// TIA Portal V18 export
// export: Created 2023-08-22T11:16:04.1404114Z, ExportSetting WithDefaults, DisplayName Totally Integrated Automation Portal, DisplayVersion V18 Update 2, DisplayName TIA Portal Openness, DisplayVersion V18 Update 2, DisplayName TIA Portal Version Control Interface, DisplayVersion V18, DisplayName SINAMICS Startdrive Advanced, DisplayVersion V18, DisplayName SINAMICS Startdrive G130, G150, S120, S150, SINAMICS MV, S210, DisplayVersion V18, DisplayName SINAMICS Startdrive G110M, G120, G120C, G120D, G120P, G115D, DisplayVersion V18, DisplayName STEP 7 Professional, DisplayVersion V18 Update 2, DisplayName STEP 7 Safety, DisplayVersion V18, DisplayName WinCC Advanced / Unified PC, DisplayVersion V18 Update 2
TYPE "typeSinaSpeedInterface"
// stored: IsFailsafeCompliant false
   STRUCT
      control : Struct
         enableAxis : Bool;
         ackError : Bool;
         speedSp : Real;
         refSpeed : Real;
         configAxis : Word := 16#003F;
         hwidStw : HW_SUBMODULE;
         hwidZsw : HW_SUBMODULE;
      END_STRUCT;
      status : Struct
         axisEnabled : Bool;
         lockout : Bool;
         actVelocity : Real;
         error : Bool;
         status : Int;
         diagId : Word;
      END_STRUCT;
   END_STRUCT;
END_TYPE
